{attribute addProperty BoxType "EPP3204-0002-0016"}
{attribute addProperty Id "RTD_RTDInputs_ChannelAT %I*ARRAY[0..6] OF RTD_RTDInputs_Channel_4364CDB6296370WcStateAT %I*WcState_98A4DF7520.250InfoDataAT %I*InfoData_BC63D37F80100"}
{attribute addProperty CRC "316216872"}
{attribute addProperty SizeInBites "378"}
{attribute addProperty SizeInBytes "47.25"}
TYPE EPP3204_72ABB954 :
STRUCT
	{attribute addProperty Name "RTD_RTDInputs_Channel"}
	RTD_RTDInputs_Channel : ARRAY[0..6] OF RTD_RTDInputs_Channel_4364CDB6;
	{attribute addProperty Name "WcState"}
	WcState : WcState_98A4DF75;
	{attribute addProperty Name "InfoData"}
	InfoData : InfoData_BC63D37F;
END_STRUCT
END_TYPE

(* stored: Version 1.2.0.0, ProductVersion 3.1.4024.9
   DUT EPP3204_72ABB954: Id {ae6795be-233b-4454-9962-f949f74588ac} *)
